{attribute 'linkalways'} 
{attribute 'no_explicit_call' := 'This FB is a CLASS and must be accessed using methods or properties'}
{attribute 'enable_dynamic_creation'}
FUNCTION_BLOCK Node_F_VN_DecomposeAffineTransformation EXTENDS VisionNode
VAR
    aAffineTransform : _TcVnMatrix2x3_LREAL;
    fRotationAngle : _LREAL(0.0);
    hrPrev : _HRESULT(S_OK);
	hresult : _HRESULT(S_OK);
END_VAR

METHOD PUBLIC  Clone : I_Node
VAR
	pNode : POINTER TO Node_F_VN_DecomposeAffineTransformation;
END_VAR
pNode := __NEW(Node_F_VN_DecomposeAffineTransformation);
Clone := pNode^;
END_METHOD

METHOD FB_init : BOOL
VAR_INPUT
	bInitRetains : BOOL; // if TRUE, the retain variables are initialized (warm start / cold start)
	bInCopyCode : BOOL;  // if TRUE, the instance afterwards gets moved into the copy code (online change)
END_VAR
AddInput('aAffineTransform', aAffineTransform);
AddInput('hrPrev', hrPrev);
AddOutput('fRotationAngle', fRotationAngle);
AddOutput('hresult',hresult);
END_METHOD

METHOD PROTECTED OnExecute
hresult.Value := F_VN_DecomposeAffineTransformation(
	aAffineTransform := aAffineTransform.Value, 
	fRotationAngle := fRotationAngle.Value, 
	hrPrev := hrPrev.Value);
END_METHOD

METHOD PUBLIC PreExecutionCheck
VAR_INPUT
	Check : I_PreExecutionChecks;
END_VAR
END_METHOD

END_FUNCTION_BLOCK

(* stored: Version 1.1.0.1, ProductVersion 3.1.4024.13
   POU Node_F_VN_DecomposeAffineTransformation: Id {3e630637-5e61-0823-17a1-018d02e335a8}, SpecialFunc None
   Folder Constructor: Id {cbcbef39-b7a9-0ca2-11ea-c7792dac5fa8}
   Method Clone: Id {275c6ae5-e00f-0610-264f-cdc8583de0d1}
   Method FB_init: Id {04b03df8-1a5b-05af-0294-ed88fc185e61}
   Method OnExecute: Id {1a73cdae-c91a-0981-22b1-201ceb9ee4b2}
   Method PreExecutionCheck: Id {fd9ab8a6-fb36-06cd-0844-ccb5c0a1b78d} *)
